FUNCTION_BLOCK FB_PowerAll
VAR_INPUT
	bEnable : BOOL;
END_VAR
VAR_OUTPUT
	bStatus : BOOL;
	bError : BOOL;
END_VAR
VAR
	power1 : MC_Power;
	power2 : MC_Power;
END_VAR
VAR_IN_OUT
	io_M1 : AXIS_REF;
	io_M2 : AXIS_REF;
END_VAR

power1(Axis := io_M1, Enable := bEnable, Enable_Negative := bEnable, Enable_Positive := bEnable);
power2(Axis := io_M2, Enable := bEnable, Enable_Negative := bEnable, Enable_Positive := bEnable);

bError := power1.Error OR power2.Error;
bStatus := power1.Status AND power2.Status AND NOT bError;

END_FUNCTION_BLOCK

(* stored: Version 1.1.0.1, ProductVersion 3.1.4024.9
   POU FB_PowerAll: Id {2e910ecb-c84c-412d-bd36-a31fe2d44037}, SpecialFunc None *)
